TYPE TcoUrRobotics_T2O_Joints_IO :
STRUCT
    bArray AT %I* : ARRAY[0..103] OF BYTE;
END_STRUCT
END_TYPE

(* stored: Version 1.1.0.1, ProductVersion 3.1.4024.12
   DUT TcoUrRobotics_T2O_Joints_IO: Id {5e225963-8293-003a-04ee-7234ea3a9966} *)
